// TIA Portal V20 export
DATA_BLOCK "IDB_LineB1"   // DB9
// stored: InstanceOfName LineB1.FB_LineB1, InstanceOfType FB, Namespace LineB1
"LineB1.FB_LineB1"
   // VAR
   //    "Conveyor_B1.1.1" : "Global.FB_Conveyor";
   //    "MABS_B1.1.1" : "Global.FB_MABS";
   //    "Transfer_B1.1.1" : "Global.FB_S300_tTransMode";
   //    "Transfer_B1.1.2" : "LineB1.FB_S300_FullControl";
   // END_VAR
BEGIN
END_DATA_BLOCK
